(* PLC project Unnamed, Unknown Unnamed 1 *)
(* stored: creationDateTime 2024-10-22T20:46:28, modificationDateTime 2024-10-24T23:57:50 *)

PROGRAM Humus
  VAR
    FilterPresureSwitchHigh AT %IX0.15 : INT;
    FilterPressureSwitchLow AT %IX0.16 : INT;
    RoughingTricklingFilterVolume AT %MW0.0 : INT := 1063 M^3;
    RoughingCircularHumusTank AT %MW0.1 : INT := 144.3 M^2;
    SludgePumpControl AT %QX0.5 : BOOL;
    MixerControl AT %QX0.6 : BOOL;
    FilterFlowControlvalve AT %QX0.8 : BOOL;
    FilterationControl AT %QX0.16 : BOOL;
  END_VAR

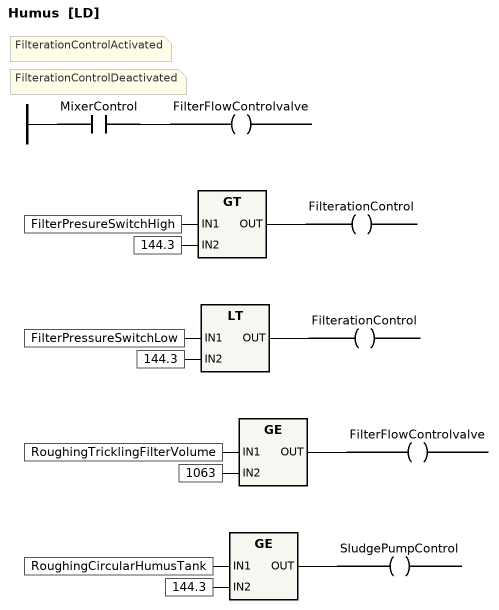
(* LD diagram, written out as Structured Text *)
(* FilterationControlDeactivated *)
FilterationControl := FilterPresureSwitchHigh > 144.3;
(* FilterationControlActivated *)
FilterationControl := FilterPressureSwitchLow < 144.3;
FilterFlowControlvalve := RoughingTricklingFilterVolume >= 1063;
FilterFlowControlvalve := MixerControl;
SludgePumpControl := RoughingCircularHumusTank >= 144.3;
END_PROGRAM

CONFIGURATION Config0
  RESOURCE Res0 ON PLC
    TASK task0(INTERVAL := T#20ms, PRIORITY := 0);
    PROGRAM instance0 WITH task0 : Humus;
  END_RESOURCE
END_CONFIGURATION
